TYPE AX5000_P_0278 :
STRUCT
	Ignore_for_one_PreOp_SafeOp_transition:UINT;
END_STRUCT
END_TYPE

(* stored: Version 1.1.0.1, ProductVersion 3.1.4024.3
   DUT AX5000_P_0278: Id {1d37709d-dcdb-49a2-919e-9b6fc8bea0c9} *)
